// TIA Portal V15.1 export
// export: Created 2023-01-03T10:05:14.5467529Z, ExportSetting None, DisplayName Totally Integrated Automation Portal, DisplayVersion V15.1 Update 5, DisplayName TIA Portal Openness, DisplayVersion V15.1 Update 5, DisplayName TIA Portal Teamcenter Gateway, DisplayVersion V15.1 Update 5, DisplayName SINAMICS Startdrive Advanced, DisplayVersion V15.1, DisplayName G130, G150, S120, S150, SINAMICS MV, S210, DisplayVersion V15.1, DisplayName G110M, G120, G120C, G120D, G120P, DisplayVersion V15.1, DisplayName STEP 7 Professional, DisplayVersion V15.1 Update 5, DisplayName Soft Starter ES, DisplayVersion V15.1, DisplayName WinCC Professional, DisplayVersion V15.1 Update 5, DisplayName SIMATIC Visualization Architect, DisplayVersion V15.1
VAR_GLOBAL   // PLC tag table "Додатково (PSL_SAF_)__PF_H1"
   I_PF_H1_001KV1_24_PSL400 AT %I0.0 : Bool;   // Додатково| =PF+H1#001_KV1--->=PF+H2_A100:1//Ввід силовий: Напруга 400VAC ок
   I_PF_H1_001QF1_4_PSL400 AT %I0.1 : Bool;   // Додатково| =PF+H1#001_QF1--->=PF+H2_A100:5//Ввід силовий: Вхідний автомат силового живлення
   I_PF_H1_003QF1_1_54_PSL230 AT %I0.2 : Bool;   // Додатково| =PF+H1#003_QF1--->=PF+H2_A100:2//Оперативні кола 230 VAC: Живлення трансформатору оперативних кіл 230 VAC
   I_PF_H1_003QF2_14_PSL230 AT %I0.3 : Bool;   // Додатково| =PF+H1#003_QF2--->=PF+H2_A100:6//Оперативні кола 230 VAC: Живлення оперативної напруги 230 VAC
   I_PF_H1_003F1_14_PSL230 AT %I1.0 : Bool;   // Додатково| =PF+H1#003_F1--->=PF+H2_A101:1//Оперативні кола 230 VAC: Живлення оперативної напруги 24VDC
   I_PF_H1_003F2_14_PSL230 AT %I1.1 : Bool;   // Додатково| =PF+H1#003_F2--->=PF+H2_A101:5//Оперативні кола 230 VAC: Живлення кіл безпеки
   I_PF_H1_003F3_14_PSL230 AT %I1.2 : Bool;   // Додатково| =PF+H1#003_F3--->=PF+H2_A101:2//Оперативні кола 230 VAC: Живлення котушок контакторів
   I_PF_H1_004T1_14_PSL24 AT %I1.3 : Bool;   // Додатково| =PF+H1#004_T1--->=PF+H2_A101:6//Оперативні кола 24 VDC: 24 VDC OK
   I_PF_H1_004QF1_14_PSL24 AT %I2.0 : Bool;   // Додатково| =PF+H1#004_QF1--->=PF+H2_A102:1//Оперативні кола 24 VDC: Живлення оперативної напруги 24VDC
   I_PF_H1_004F1_14_PSL24 AT %I2.1 : Bool;   // Додатково| =PF+H1#004_F1--->=PF+H2_A102:5//Оперативні кола 24 VDC: Живлення реле безпеки
   I_PF_H1_004F2_14_PSL24 AT %I2.2 : Bool;   // Додатково| =PF+H1#004_F2--->=PF+H2_A102:2//Оперативні кола 24 VDC: Живлення модулів DO/AO
   I_PF_H1_004F5_14_PSL24 AT %I2.3 : Bool;   // Додатково| =PF+H1#004_F5--->=PF+H2_A102:6//Оперативні кола 24 VDC: Живлення котушок клапанів зони загрузки
   I_PF_H1_004F6_14_PSL24 AT %I3.0 : Bool;   // Додатково| =PF+H1#004_F6--->=PF+H2_A103:1//Оперативні кола 24 VDC: Живлення котушок клапанів зони розгрузки
   I_PF_H1_004UPS1_1_PSL24 AT %I3.1 : Bool;   // Додатково| =PF+H1#004_UPS1--->=PF+H2_A103:5//Оперативні кола 24 VDC: БЛОК безперебійного електроживлення BAT.
   I_PF_H1_004UPS1_4_PSL24 AT %I3.2 : Bool;   // Додатково| =PF+H1#004_UPS1--->=PF+H2_A103:2//Оперативні кола 24 VDC: БЛОК безперебійного електроживлення ALARM
   I_PF_H1_004F10_14_PSL24 AT %I3.3 : Bool;   // Додатково| =PF+H1#004_F10--->=PF+H2_A103:6//Оперативні кола 24 VDC: Живлення шафи Т1 (Станція ET200)
   I_PF_H1_004F11_14_PSL24 AT %I4.0 : Bool;   // Додатково| =PF+H1#004_F11--->=PF+H2_A104:1//Оперативні кола 24 VDC: Живлення шафи Т2 (Панель оператора)
   I_PF_H1_004F12_14_PSL24 AT %I4.1 : Bool;   // Додатково| =PF+H1#004_F12--->=PF+H2_A104:5//Оперативні кола 24 VDC: Живлення шафи Т3 (Станція ET200)
   I_PF_H1_005SB1_4_SAF AT %I4.2 : Bool;   // Додатково| =PF+H1#005_SB1--->=PF+H2_A104:2//Кола безпеки: Аварійний стоп
   I_PF_H1_005SB2_4_SAF AT %I4.3 : Bool;   // Додатково| =PF+H1#005_SB2--->=PF+H2_A104:6//Кола безпеки: Квітувати аварію
   I_PF_H1_005KM2_14_SAF AT %I5.0 : Bool;   // Додатково| =PF+H1#005_KM2--->=PF+H2_A105:1//Кола безпеки: Контактори кіл безпеки
   I_PF_H1_005KM3_34_SAF AT %I5.1 : Bool;   // Додатково| =PF+H1#005_KM3--->=PF+H2_A105:5//Кола безпеки: ЗЗ Подати напругу
   Q_PF_H1_005KL1__A1_SAF AT %Q0.0 : Bool;   // Додатково| =PF+H1#005_KL1--->=PF+H2_A200:1//Кола безпеки: Квітування реле безпеки
   Q_PF_H1_005SB2_x1_SAF AT %Q0.1 : Bool;   // Додатково| =PF+H1#005_SB2--->=PF+H2_A200:5//Кола безпеки: Квітувати аварію
   Q_PF_H1_005HL1_x1_SAF AT %Q0.2 : Bool;   // Додатково| =PF+H1#005_HL1--->=PF+H2_A200:2//Кола безпеки: Напругу подано
END_VAR
